// Buttons control logic
FUNCTION_BLOCK PUBLIC InterfaceControlPanel
VAR_INPUT
	StartButton : BOOL;
	ResetButton : BOOL;
	StopButton : BOOL;
	blink : BOOL;
END_VAR
VAR_IN_OUT
	isStopON : BOOL;
	isSystemON : BOOL;
	isResetON : BOOL;
END_VAR
VAR_OUTPUT
	StartLight : BOOL;
	StopLight : BOOL;
	ResetLight : BOOL;
END_VAR
VAR
END_VAR

// Memory bit for isSystemON
IF StartButton THEN
	isSystemON := TRUE;
END_IF;

IF NOT StopButton THEN
	isSystemON := FALSE;
END_IF;
// -------------
// Memory bit for isStopON
IF NOT StopButton THEN
	isStopON := TRUE;
END_IF;

IF isSystemON THEN
	isStopON := FALSE;
END_IF;
// -------------
// Memory bit for isResetON
IF ResetButton THEN
	isResetON := TRUE;
END_IF;

IF isSystemON THEN
	isResetON := FALSE;
END_IF;
// -------------
// ------------- OUTPUTS ---------------
StartLight := isSystemON OR (isStopON AND NOT isSystemON AND blink);
//
ResetLight := isResetON;
//
StopLight := isStopON AND NOT isSystemON;

END_FUNCTION_BLOCK

(* stored: Version 1.1.0.1, ProductVersion 3.1.4024.12
   POU InterfaceControlPanel: Id {27c35da5-f9a5-42cc-a2e3-c07c15751685}, SpecialFunc None *)
